Universal Robots PolyScope program: motor_plate_positioning.urp

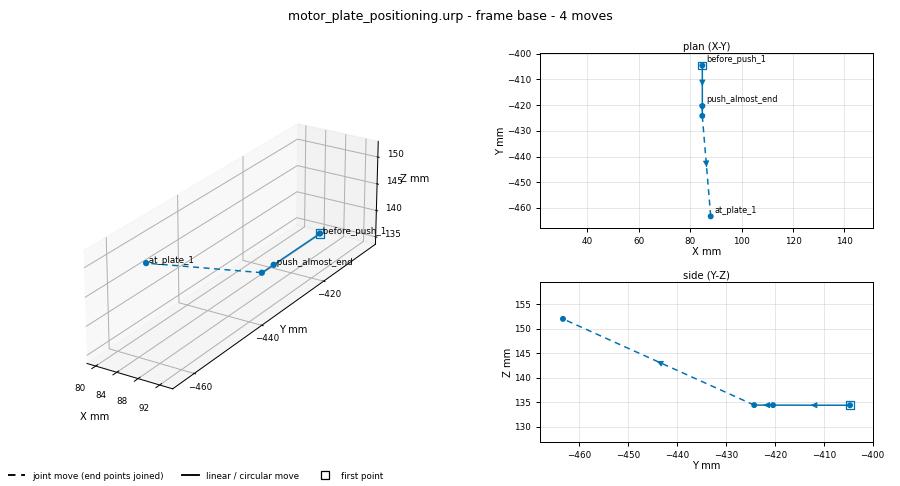
[picture p0: tool path of motor_plate_positioning.urp in frame base, 4 of 4 moves have a stored position in this frame; points joined in program order, loops and branches not executed]
Program motor_plate_positioning (installation=default directory=/programs/wrs2020 createdIn=5.9.1.1031110 lastSavedIn=5.9.1.1031110 robotSerialNumber=20205500180)
Calibrated DH parameters: a=[0, -0.425, -0.3922, 0, 0, 0]; d=[0.1625, 0, 0, 0.1333, 0.0997, 0.0996]; alpha=[1.570796, 0, 0, 1.570796, -1.570796, 0]; deltaTheta=[0, 0, 0, 0, 0, 0]
Robot Program (runOnlyOnce=true)
  MoveL speed 250 mm/s, acceleration 1200 mm/s^2 (useActiveTCP=false) tcp=gripper_140_tip; feature=Base
    Waypoint before_push_1: TCP in base x=84.741 y=-404.629 z=134.416 mm, rx=0.0046 ry=-3.002 rz=0.8772 rad; joints [78.516, -122.292, 148.167, -148.053, -84.559, -10.089] deg; TCP offset x=0 y=0 z=220 mm, rx=0 ry=0 rz=0 rad
  URCap Gripper (Robotiq_Grippers, Robotiq Inc.) dataModel(position=100.0, force=0.0, speed=0.0, positionInDouble=100.0, forceInDouble=0.0, speedInDouble=0.0, slaveIds=[9], blocking=true)
  MoveL speed 250 mm/s, acceleration 1200 mm/s^2 (useActiveTCP=false) tcp=gripper_140_tip; feature=Base
    Waypoint push_almost_end: motionParameters(jointSpeed=1.047198 jointAcceleration=1.396263 cartesianSpeed=0.1 cartesianAcceleration=0.1 blendRadius=0.002); TCP in base x=84.751 y=-420.361 z=134.44 mm, rx=0.0046 ry=-3.002 rz=0.8773 rad; joints [79.309, -118.419, 146.69, -150.515, -84.981, -9.415] deg
    Waypoint push_end_1: motionParameters(jointSpeed=1.047198 jointAcceleration=1.396263 cartesianSpeed=0.05 cartesianAcceleration=0.008); TCP in base x=84.73 y=-424.199 z=134.446 mm, rx=0.0045 ry=-3.002 rz=0.8773 rad; joints [79.484, -117.517, 146.313, -151.054, -85.077, -9.264] deg
    SuppressedNode
      Waypoint before_push_2: motionParameters(jointSpeed=1.047198 jointAcceleration=1.396263 cartesianSpeed=0.8 cartesianAcceleration=0.8); TCP in base x=88.017 y=-382.896 z=133.609 mm, rx=0.004 ry=3.1409 rz=-0.0122 rad; joints [83.034, -104.382, 122.465, -108.52, -89.91, -6.818] deg
  URCap Gripper (Robotiq_Grippers, Robotiq Inc.) dataModel(position=70.19607843137254, force=100.0, speed=100.0, positionInDouble=70.19607843137254, forceInDouble=100.0, speedInDouble=100.0, slaveIds=[9], blocking=true)
  MoveJ speed 150 deg/s, acceleration 150 deg/s^2 (useActiveTCP=false) tcp=gripper_140_tip; feature=Base
    SuppressedNode
      Waypoint above_plate_1: motionParameters(blendRadius=0.03); TCP in base x=88.01 y=-440.155 z=173.172 mm, rx=0.0038 ry=3.0942 rz=-0.5374 rad; joints [81.985, -110.774, 128.458, -127.209, -87.271, -7.405] deg
    Waypoint at_plate_1: TCP in base x=88.005 y=-463.265 z=152.055 mm, rx=0.0034 ry=2.946 rz=-1.087 rad; joints [79.411, -112.569, 147.397, -164.842, -83.11, -7.945] deg
  URCap Gripper (Robotiq_Grippers, Robotiq Inc.) dataModel(position=100.0, force=0.0, speed=0.0, positionInDouble=100.0, forceInDouble=0.0, speedInDouble=0.0, slaveIds=[9], blocking=true)
  URCap Gripper (Robotiq_Grippers, Robotiq Inc.) dataModel(position=82.3529411764706, force=100.0, speed=0.0, positionInDouble=82.3529411764706, forceInDouble=100.0, speedInDouble=0.0, slaveIds=[9], blocking=true)
